# B&R Automation Studio project EFI (part 26)

#### CleaningTests.c - Groups test cases for addition
```c
/********************************************************************
 * COPYRIGHT -- Bernecker + Rainer
 ********************************************************************
 * Program: ConsentsTests
 * Author: Jorge Murria
 ********************************************************************
 * Prepare machine with basic test to allow proper behabior
 * and starting tasks
 ********************************************************************/

#include <bur/plctypes.h>

#ifdef _DEFAULT_INCLUDES
#include <AsDefault.h>
#endif

#include "UnitTest.h"

#include <stdio.h>
#include <unistd.h>
#include <time.h>         /* clock_t, clock, CLOCKS_PER_SEC */

_LOCAL TIME TimeLast;
_LOCAL TIME endtime;
_LOCAL UDINT diff_t;
_LOCAL STRING stringAux[120];

#define FALSE 0
#define TRUE 1

_LOCAL UDINT previousTileCounter;

void nextState(){
	exTimesPreFast = gMachine.St.exec.fast;
	exTimesPreSlow = gMachine.St.exec.slow;
	iTestState++;
	TimeLast = clock_ms();
	diff_t = diff_t;
	stringAux[120] = stringAux[120];
}

_TEST test_ReturningToPrint(void)
{
	strcpy(txTest, "test_ReturningToPrint");
	switch (iTestState)
	{
		case 0:
			gSimMachine.Commands.xToZero = TRUE;
			gFeeder.ParSw.xEnabled=FALSE;
			gPrimer.ParSw.xEnabled=FALSE;
			gDryerAnc.ParSw.xEnabled=FALSE;
			gStacker.ParSw.xEnabled=FALSE;
			gMachine.parSw.Media.rLength = 1600;
			gSimThickCtrl.Commands.xEmptyMediaTracking = TRUE;
			nextState();
			break;

		case 1:
			strcpy(txStateDesc, "Waiting the machine to be in Zero");
			TEST_BUSY_CONDITION( !gMachine.St.Mode.xZero );
			nextState();
			break;

		case 2:
			gSimMachine.Commands.xToAuto = TRUE;
			nextState();
			break;

		case 3:
			strcpy(txStateDesc, "Waiting the machine to be in Auto");
			TEST_BUSY_CONDITION( !gMachine.St.Mode.xAuto );
			TEST_BUSY_CONDITION( gMachine.St.exec.fast < exTimesPreFast + 8 ); //We'll wait xx scan cycles
			TEST_BUSY_CONDITION( !gMachine.St.Position.xInCap );
			gSimMachine.Commands.xToProduction = TRUE;
			nextState();
			break;

		case 4:
			strcpy(txStateDesc, "Going to Production");
			TEST_BUSY_CONDITION( !gMachine.St.AutoMode.xProduction);
			gMachine.commandsSw.xStart_GI = FALSE;
			nextState();
			break;

		case 5:
			strcpy(txStateDesc, "Waiting to be GoingToPrint");
			TEST_BUSY_CONDITION( !gMachine.St.Position.xGoingToPrint );
			TEST_BUSY_CONDITION( gBlock[1].Status.rMotorPosition > gBlock[1].parameters.Motor.rDripBarsPosition - 10);
			nextState();
			break;

		case 6:
			strcpy(txStateDesc, "Order to Clean");
			if(!gMachine.Pt.xControlledByLine ){
				gBlock[1].commands.xForceCleanNoDelay = TRUE;
			}
			else{
				gLine.Commands.Clean = TRUE;
			}
			TEST_BUSY_CONDITION( !gBlock[1].Status.Position.xCleaning);
			nextState();
			break;

		case 7:
			strcpy(txStateDesc, "Waiting to remove the signal");
			TEST_BUSY_CONDITION( gMachine.St.exec.fast < exTimesPreFast + 3 ); //We'll wait xx scan cycles
			gBlock[1].commands.xForceCleanNoDelay = FALSE;
			nextState();
			break;

		case 8:
			strcpy(txStateDesc, "Waiting to start cleaning");
			TEST_BUSY_CONDITION(gBlock[1].Status.Position.xCleaning); //We'll wait xx scan cycles
			nextState();
			break;

		case 9:
			strcpy(txStateDesc, "Waiting to finish cleaning");
			TEST_BUSY_CONDITION( gBlock[1].Status.rMotorPosition > gBlock[1].parameters.Motor.rDripBarsPosition - 10);
			nextState();
			break;

		case 10:
			endtime = clock_ms();
			TEST_BUSY_CONDITION( endtime < TimeLast + 2000 ); //We'll wait xx ms
			//TEST_ASSERT(gBlock[1].Status.Position.xGoingToPrint || gBlock[1].Status.Position.xInPrint); //If variable is TRUE, the test is correct
			TEST_ASSERT(!gBlock[1].Status.Position.xCleaning);
			nextState();
			break;

		case 11:
			strcpy(txStateDesc, "Check activation of waste ink pump");
			if(gBlock[1].parameters.xWastedInkTankProcess){
				TEST_ASSERT(gBlock[1].Out.xWastedInkTankPump);
			}

			iTestState = 0;
			TEST_DONE;

			break;

		default:
			break;
	}
}

_TEST test_ReturningToCap(void)
{
	strcpy(txTest, "test_ReturningToCap");
	switch (iTestState)
	{
		case 0:
			gSimMachine.Commands.xToZero = TRUE;
			gSimThickCtrl.Commands.xEmptyMediaTracking = TRUE;
			nextState();
			break;

		case 1:
			strcpy(txStateDesc, "Waiting the machine to be in Zero");
			TEST_BUSY_CONDITION( !gMachine.St.Mode.xZero );
			nextState();
			break;

		case 2:
			endtime = clock_ms();
			TEST_BUSY_CONDITION( endtime < TimeLast + 100 ); //We'll wait xx ms
			gSimMachine.Commands.xToAuto = TRUE;
			nextState();
			break;

		case 3:
			strcpy(txStateDesc, "Waiting the machine to be in Auto");
			TEST_BUSY_CONDITION( !gMachine.St.Mode.xAuto );
			nextState();
			break;

		case 4:
			strcpy(txStateDesc, "Waiting to be in Cap or GoingToCap");
			TEST_BUSY_CONDITION( gMachine.St.exec.fast < exTimesPreFast + 3 ); //We'll wait xx scan cycles
			TEST_BUSY_CONDITION( !gBlock[1].Status.Position.xGoingToCap  && !gBlock[1].Status.Position.xInCap);
			nextState();
			break;

		case 5:
			TEST_BUSY_CONDITION(!gBlock[1].Status.Position.xInCap);
			nextState();
			break;

		case 6:
			strcpy(txStateDesc, "Order to Clean");
			if(!gMachine.Pt.xControlledByLine ){
				gBlock[1].commands.xForceCleanNoDelay = TRUE;
			}
			else{
				gLine.Commands.Clean = TRUE;
			}
			TEST_BUSY_CONDITION( !gBlock[1].Status.Position.xCleaning); //We'll wait xx scan cycles
			nextState();
			break;

		case 7:
			strcpy(txStateDesc, "Waiting to remove the signal");
			TEST_BUSY_CONDITION( gMachine.St.exec.fast < exTimesPreFast + 3 ); //We'll wait xx scan cycles
			gBlock[1].commands.xForceCleanNoDelay = FALSE;
			nextState();
			break;

		case 8:
			strcpy(txStateDesc, "Waiting to start cleaning");
			TEST_BUSY_CONDITION( !gBlock[1].Status.Position.xCleaning); //We'll wait xx scan cycles
			nextState();
			break;

		case 9:
			strcpy(txStateDesc, "Waiting to finish cleaning");
			TEST_BUSY_CONDITION( gBlock[1].Status.Position.xCleaning); //We'll wait xx scan cycles
			nextState();
			break;

		case 10:
			TEST_BUSY_CONDITION( gMachine.St.exec.fast < exTimesPreFast + 3 ); //We'll wait xx scan cycles
			TEST_ASSERT(gBlock[1].Status.Position.xGoingToCap || gBlock[1].Status.Position.xInCap); //If variable is TRUE, the test is correct

			iTestState = 0;
			TEST_DONE;

			break;

		default:
			break;
	}
}

_TEST test_CheckAnyCleaningModeIsEnabled(void)
{
	strcpy(txTest, "test_CheckAnyCleaningModeIsEnabled");
	switch (iTestState)
	{
		case 0:
			gSimMachine.Commands.xToZero = TRUE;
			gMachine.parSw.Clean.xCleanSystemByPieces = FALSE;
			gMachine.parSw.Clean.xCleanSystemByTime = FALSE;
			gSimThickCtrl.Commands.xEmptyMediaTracking = TRUE;
			nextState();
			break;

		case 1:
			strcpy(txStateDesc, "Waiting to finish cleaning");
			TEST_BUSY_CONDITION( gMachine.St.exec.fast < exTimesPreFast + 8 ); //We'll wait xx scan cycles
			TEST_ASSERT(gMachine.Al.Warning.xNoCleaningModeEnabled); //If variable is TRUE, the test is correct

			iTestState = 0;
			TEST_DONE;

			break;

		default:
			break;
	}
}

_TEST test_CleaningByTilesTwice(void)
{
	//If the Test makes non sense, not execute it.
	if (gMachine.Pt.PDSignalTpe==PDCFG_SENSOR){

		iTestState = 0;
		TEST_DONE;
	}
	strcpy(txTest, "test_CleaningByTilesTwice");
	switch (iTestState)
	{
		case 0:
			gSimMachine.Commands.xToZero = TRUE;
			gMachine.parSw.Clean.xCleanSystemByPieces = TRUE;
			gSimMachine.Signals.xPDCarriageSignalL1 = FALSE; //To be sure to receive later the required edge
			gMachine.parSw.Clean.iPiecesNumberToCleanL1 = 10;
			gMachine.parSw.Clean.tiTimeDelayToCleanL1 = 1000;
			gMachine.parSw.Clean.tiTimeDelayGapToClean = 1000;
			gSimThickCtrl.Commands.xEmptyMediaTracking = TRUE;
			nextState();
			break;

		case 1:
			strcpy(txStateDesc, "Waiting the machine to be in Zero");
			TEST_BUSY_CONDITION( !gMachine.St.Mode.xZero );
			nextState();
			break;

		case 2:
			endtime = clock_ms();
			TEST_BUSY_CONDITION( endtime < TimeLast + 100 ); //We'll wait xx ms
			gSimMachine.Commands.xToAuto = TRUE;
			nextState();
			break;

		case 3:
			strcpy(txStateDesc, "Waiting the machine to be in Auto");
			TEST_BUSY_CONDITION( !gMachine.St.Mode.xAuto );
			nextState();
			break;

		case 4:
			strcpy(txStateDesc, "Waiting to be in Cap or GoingToCap");
			TEST_BUSY_CONDITION( gMachine.St.exec.fast < exTimesPreFast + 3 ); //We'll wait xx scan cycles
			TEST_BUSY_CONDITION( !gBlock[1].Status.Position.xGoingToCap  && !gBlock[1].Status.Position.xInCap);
			gMachine.commandsSw.xToNormal_GI = TRUE;
			nextState();
			break;

		case 5:
			strcpy(txStateDesc, "Waiting to be in Production");
			TEST_BUSY_CONDITION( !gMachine.St.AutoMode.xProduction );
			TEST_BUSY_CONDITION( gMachine.St.exec.fast < exTimesPreFast + 20 ); //We'll wait xx scan cycles
			gSimMachine.Commands.xToProduction = TRUE;
			gMachine.commandsSw.xToNormal_GI = FALSE;
			nextState();
			break;

		case 6:
			TEST_BUSY_CONDITION( gMachine.St.exec.fast < exTimesPreFast + 20 ); //We'll wait xx scan cycles
			gMachine.commandsSw.xStart_GI = FALSE;
			TEST_BUSY_CONDITION( !gBelt.states.xRuningBelt );
			previousTileCounter = gMachine.Lg.udiPiecesCounterL1;
			gDing.In.xDingLow = TRUE;
			gDing.In.rHighDingMm = 5.0;
			nextState();
			break;

		case 7:
			strcpy(txStateDesc, "Raising product detects when the belt running");
			endtime = clock_ms();
			TEST_BUSY_CONDITION( endtime < TimeLast + 200 ); //We'll wait xx ms
			if(gMachine.Pt.PDSignalTpe==PDCFG_SENSOR){
				gSimMachine.Commands.Media.xContinuousMediaPresent = TRUE;
			}
			else{
				if (previousTileCounter == gMachine.Lg.udiPiecesCounterL1) {
					gSimMachine.Signals.xPDCarriageSignalL1 = TRUE;
					gSimMachine.Signals.xProductDetectL1 = TRUE;
				}
				else {
					TimeLast = clock_ms();
					previousTileCounter = gMachine.Lg.udiPiecesCounterL1;
					gSimMachine.Signals.xPDCarriageSignalL1 = FALSE;
					gSimMachine.Signals.xProductDetectL1 = FALSE;
				}
			}
			TEST_BUSY_CONDITION( !gMachine.AutoCmd.xCleanningByPiecesL1);
			gSimMachine.Commands.Media.xContinuousMediaPresent = FALSE;
			nextState();
			break;
		case 8:
			strcpy(txStateDesc, "Waiting to start cleaning");
			gDing.In.xDingLow = FALSE;
			gDing.In.rHighDingMm = 0.0;
			TEST_BUSY_CONDITION( !gBlock[1].Status.Position.xCleaning);
			nextState();
			break;

		case 9:
			strcpy(txStateDesc, "Waiting to finish cleaning");
			TEST_BUSY_CONDITION( !gBlock[1].Status.Position.xInPrint); //We'll wait xx scan cycles
			gDing.In.xDingLow = TRUE;
			gDing.In.rHighDingMm = 5.0;
			nextState();
			break;

		case 10:
			strcpy(txStateDesc, "Raising product detects 2nd round");
			TEST_BUSY_CONDITION( !gBelt.states.xRuningBelt ); //We'll wait xx scan cycles
			endtime = clock_ms();
			TEST_BUSY_CONDITION( endtime < TimeLast + 200 ); //We'll wait xx ms
			if (previousTileCounter == gMachine.Lg.udiPiecesCounterL1) {
				gSimMachine.Signals.xPDCarriageSignalL1 = TRUE;
				gSimMachine.Signals.xProductDetectL1 = TRUE;
			}
			else {
				TimeLast = clock_ms();
				previousTileCounter = gMachine.Lg.udiPiecesCounterL1;
				gSimMachine.Signals.xPDCarriageSignalL1 = FALSE;
				gSimMachine.Signals.xProductDetectL1 = FALSE;
			}
			TEST_BUSY_CONDITION( !gMachine.AutoCmd.xCleanningByPiecesL1); //We'll wait xx scan cycles
			gSimMachine.Signals.xPDCarriageSignalL1 = FALSE;
			gSimMachine.Signals.xProductDetectL1 = FALSE;
			nextState();
			break;
		case 11:
			strcpy(txStateDesc, "Waiting to start cleaning");
			gDing.In.xDingLow = FALSE;
			gDing.In.rHighDingMm = 0.0;
			TEST_BUSY_CONDITION( !gBlock[1].Status.Position.xCleaning);
			nextState();
			break;

		case 12:
			strcpy(txStateDesc, "Waiting to finish cleaning");
			TEST_BUSY_CONDITION( gBlock[1].Status.Position.xCleaning); //We'll wait xx scan cycles
			nextState();
			break;

		case 13:
			TEST_BUSY_CONDITION( gMachine.St.exec.fast < exTimesPreFast + 5 ); //We'll wait xx scan cycles
			TEST_ASSERT(gBlock[1].Status.Position.xGoingToPrint || gBlock[1].Status.Position.xInPrint); //Prior to cleaning, it was in production, in printin
			gMachine.parSw.Clean.xCleanSystemByPieces = FALSE;
			iTestState = 0;
			TEST_DONE;

			break;

		default:
			break;
	}
}

/* --- Test for DELOREAN-2123 Cleaning belt process stopping behaviour --- */
_TEST test_CleanBeltStop(void)
{
	//If the Test makes non sense, not execute it.
	if (!gMachine.Pt.Clean.xCleanBeltForUv || !gMachine.Pt.xControlledByLine){
		//This 2 lines just for the last TestCase
		strcpy(txTest, "test_CleanBeltForUv Finished!! Congrats!");
		strcpy(txStateDesc, "--");

		iTestState = 0;
		TEST_DONE;
	}

	strcpy(txTest, "test_CleanBeltStop");
	switch (iTestState)
	{
		case 0:
			gMachine.parSw.CleanBelt.iBeltTurns = 1;
			gSimMachine.Commands.xToZero = TRUE;
			gSimThickCtrl.Commands.xEmptyMediaTracking = TRUE;
			nextState();
			break;

		case 1:
			strcpy(txStateDesc, "Waiting the machine to be in Zero");
			TEST_BUSY_CONDITION( !gMachine.St.Mode.xZero );
			nextState();
			break;

		case 2:
			TEST_BUSY_CONDITION( gMachine.St.exec.fast < exTimesPreFast + 3 ); //We'll wait xx ms
			gSimMachine.Commands.xToAuto = TRUE;
			nextState();
			break;

		case 3:
			strcpy(txStateDesc, "Waiting the machine to be in Auto");
			TEST_BUSY_CONDITION( !gMachine.St.Mode.xAuto );
			TEST_BUSY_CONDITION( gMachine.St.exec.fast < exTimesPreFast + 8 ); //We'll wait xx scan cycles
			gMachine.In.Buttons.xReset = TRUE;
			nextState();
			break;

		case 4:
			strcpy(txStateDesc, "Waiting to be in idle to send clean bealt order");
			TEST_BUSY_CONDITION (gLine.Status != LINE_IDLE);
			gMachine.commandsSw.xCleanBelt = TRUE;
			nextState();
			break;

		case 5:
			strcpy(txStateDesc, "Check belt clean process is being executed");
			TEST_BUSY_CONDITION(gMachine.St.CleaningBelt.enState != CLN_BELT_CLEAN_CLOKWISE);
			gMachine.In.Buttons.xStop = TRUE;
			nextState();
			break;

		case 6:
			strcpy(txStateDesc, "Check belt cleaning stops");
			TEST_BUSY_CONDITION( gMachine.St.exec.fast < exTimesPreFast + 5 ); //We'll wait xx scan cycles
			gMachine.In.Buttons.xStop = FALSE;
			endtime = clock_ms();
			TEST_BUSY_CONDITION( gMachine.St.CleaningBelt.enState != CLN_BELT_ERROR);// && endtime < TimeLast + 1000);
			TEST_ASSERT( gMachine.St.CleaningBelt.enState == CLN_BELT_ERROR );
			nextState();
			break;

		case 7:
			strcpy(txStateDesc, "Check belt cleaning grafcet status goes back to ready");
			endtime = clock_ms();
			TEST_BUSY_CONDITION( gMachine.St.CleaningBelt.enState != CLN_BELT_READY_TO_CLEAN);// && endtime < TimeLast + 2000);
			TEST_ASSERT( gMachine.St.CleaningBelt.enState == CLN_BELT_READY_TO_CLEAN );

			//This 2 lines just for the last TestCase
			strcpy(txTest, "test_CleaningTests Finished!! Congrats!");
			strcpy(txStateDesc, "--");

			iTestState = 0;
			TEST_DONE;

			break;

		default:
			break;
	}
}
/* --- End test for DELOREAN-2123 --- */

_TEST test_StopBelWhenMediaDetectInClean(void)
{
	strcpy(txTest, "test_StopBelWhenMediaDetectInClean");
	switch (iTestState)
	{
		case 0:
			gSimMachine.Commands.xToZero = TRUE;
			gMachine.parSw.Clean.xCleanSystemByPieces = TRUE;
			gSimMachine.Signals.xPDCarriageSignalL1 = FALSE; //To be sure to receive later the required edge
			gMachine.parSw.Clean.iPiecesNumberToCleanL1 = 10;
			gMachine.parSw.Clean.tiTimeDelayToCleanL1 = 1000;
			gMachine.parSw.Clean.tiTimeDelayGapToClean = 1000;
			gSimThickCtrl.Commands.xEmptyMediaTracking = TRUE;
			nextState();
			break;

		case 1:
			strcpy(txStateDesc, "Waiting the machine to be in Zero");
			TEST_BUSY_CONDITION( !gMachine.St.Mode.xZero );
			nextState();
			break;

		case 2:
			endtime = clock_ms();
			TEST_BUSY_CONDITION( endtime < TimeLast + 100 ); //We'll wait xx ms
			gSimMachine.Commands.xToAuto = TRUE;
			nextState();
			break;

		case 3:
			strcpy(txStateDesc, "Waiting the machine to be in Auto");
			TEST_BUSY_CONDITION( !gMachine.St.Mode.xAuto );
			nextState();
			break;

		case 4:
			strcpy(txStateDesc, "Waiting to be in Cap or GoingToCap");
			TEST_BUSY_CONDITION( gMachine.St.exec.fast < exTimesPreFast + 3 ); //We'll wait xx scan cycles
			TEST_BUSY_CONDITION( !gBlock[1].Status.Position.xGoingToCap  && !gBlock[1].Status.Position.xInCap);
			gMachine.commandsSw.xToNormal_GI = TRUE;
			nextState();
			break;

		case 5:
			strcpy(txStateDesc, "Waiting to be in Production");
			TEST_BUSY_CONDITION( !gMachine.St.AutoMode.xProduction );
			TEST_BUSY_CONDITION( gMachine.St.exec.fast < exTimesPreFast + 20 ); //We'll wait xx scan cycles
			gSimMachine.Commands.xToProduction = TRUE;
			gMachine.commandsSw.xToNormal_GI = FALSE;
			nextState();
			break;

		case 6:
			TEST_BUSY_CONDITION( gMachine.St.exec.fast < exTimesPreFast + 20 ); //We'll wait xx scan cycles
			gMachine.commandsSw.xStart_GI = FALSE;
			TEST_BUSY_CONDITION( !gBelt.states.xRuningBelt );
			previousTileCounter = gMachine.Lg.udiPiecesCounterL1;
			gDing.In.xDingLow = TRUE;
			gDing.In.rHighDingMm = 5.0;
			nextState();
			break;

		case 7:
			strcpy(txStateDesc, "Raising product detects when the belt running");
			endtime = clock_ms();
			TEST_BUSY_CONDITION( endtime < TimeLast + 200 ); //We'll wait xx ms
			if(gMachine.Pt.PDSignalTpe==PDCFG_SENSOR){
				gSimMachine.Commands.Media.xContinuousMediaPresent = TRUE;
			}
			else{
				if (previousTileCounter == gMachine.Lg.udiPiecesCounterL1) {
					gSimMachine.Signals.xPDCarriageSignalL1 = TRUE;
					gSimMachine.Signals.xProductDetectL1 = TRUE;
				}
				else {
					TimeLast = clock_ms();
					previousTileCounter = gMachine.Lg.udiPiecesCounterL1;
					gSimMachine.Signals.xPDCarriageSignalL1 = FALSE;
					gSimMachine.Signals.xProductDetectL1 = FALSE;
				}
			}
			TEST_BUSY_CONDITION( !gMachine.AutoCmd.xCleanningByPiecesL1);
			gSimMachine.Commands.Media.xContinuousMediaPresent = FALSE;
			nextState();
			break;
		case 8:
			strcpy(txStateDesc, "Waiting to start cleaning");
			gDing.In.xDingLow = FALSE;
			gDing.In.rHighDingMm = 0.0;
			gPhotoCells.Inputs.Signals.xPhotoCells[1] = FALSE;
			TEST_BUSY_CONDITION( !gBlock[1].Status.Position.xCleaning);
			nextState();
			break;

		case 9:
			strcpy(txStateDesc, "Detect Media In");
			if (gDing.State.xDingInstalled){
				gDing.In.xDingLow = TRUE;
				gDing.In.rHighDingMm = 5.0;
			}
			else{
				gPhotoCells.Inputs.Signals.xPhotoCells[1] = TRUE;
			}
			nextState();
			break;

		case 10:
			TEST_BUSY_CONDITION( gMachine.St.exec.fast < exTimesPreFast + 10 ); //We'll wait xx scan cycles
			TEST_ASSERT(!gBelt.states.xRuningBelt); //Prior to cleaning, it was in production, in printing
			nextState();
			break;

		case 11:
			strcpy(txStateDesc, "Waiting to finish cleaning");
			TEST_BUSY_CONDITION( gBlock[1].Status.Position.xCleaning); //We'll wait xx scan cycles
			gMachine.parSw.Clean.xCleanSystemByPieces = FALSE;
			gDing.In.xDingLow = FALSE;
			gPhotoCells.Inputs.Signals.xPhotoCells[1] = FALSE;
			//This 2 lines just for the last TestCase
			strcpy(txTest, "test_CleaningTests Finished!! Congrats!");
			strcpy(txStateDesc, "--");
			iTestState = 0;
			TEST_DONE;

			break;

		default:
			break;

//		case 12:
//			TEST_BUSY_CONDITION( gMachine.St.exec.fast < exTimesPreFast + 5 ); //We'll wait xx scan cycles
//			TEST_ASSERT(gBlock[1].Status.Position.xGoingToPrint || gBlock[1].Status.Position.xInPrint); //Prior to cleaning, it was in production, in printing
//			gMachine.parSw.Clean.xCleanSystemByPieces = FALSE;
//			//This 2 lines just for the last TestCase
//			strcpy(txTest, "test_CleaningTests Finished!! Congrats!");
//			strcpy(txStateDesc, "--");
//			iTestState = 0;
//			TEST_DONE;

//			break;

//		default:
//			break;

	}
}

_TEST test_StopVenturiWhenCloseToEnd(void)
{
	strcpy(txTest, "test_StopVenturiWhenCloseToEnd");
	switch (iTestState)
	{
		case 0:
			strcpy(txStateDesc, "Preparing test conditions...");
			gSimMachine.Commands.xToZero = TRUE;
			gSimThickCtrl.Commands.xEmptyMediaTracking = TRUE;
			nextState();
			break;

		case 1:
			TEST_BUSY_CONDITION (!gMachine.St.Mode.xZero);
			gSimMachine.Commands.xToAuto = TRUE;
			nextState();
			break;

		case 2:
			TEST_BUSY_CONDITION (!gMachine.St.Mode.xAuto);
			TEST_BUSY_CONDITION( !gBlock[1].Status.Position.xInCap);
			nextState();
			break;

		case 3:
			strcpy(txStateDesc, "Giving clean order...");
			TEST_BUSY_CONDITION ( gMachine.St.exec.fast < exTimesPreFast + 20 );
			gMachine.commands.xClean = TRUE;
			nextState();
			break;

		case 4:
			strcpy(txStateDesc, "Waiting for clean procss...");
			TEST_BUSY_CONDITION (!gBlock[1].Status.Position.xCleaning);
			TEST_BUSY_CONDITION (!gBlock[1].Status.Icla.xIsMoving);
			nextState();
			break;

		case 5:
			strcpy(txStateDesc, "Venturi should turn on");
			TEST_BUSY_CONDITION ( gBlock[1].Status.Icla.rCurrentPosition <= gBlock[1].parameters.Icla.rLastHeadPosition);
			nextState();
			break;

		case 6:
			TEST_BUSY_CONDITION ( gBlock[1].Status.Icla.rCurrentPosition >= (gBlock[1].parameters.Icla.rLastHeadPosition));
			nextState();
			break;

		case 7:
			TEST_BUSY_CONDITION(gMachine.St.exec.slow < exTimesPreSlow +3);
			TEST_ASSERT(gBlock[1].Out.xVenturi);
			nextState();
			break;

		case 8:
			strcpy(txStateDesc, "Venturi should turn off");
			TEST_BUSY_CONDITION ( gBlock[1].Status.Icla.rCurrentPosition >= gBlock[1].parameters.Icla.rFirstHeadPosition);
			nextState();
			break;

		case 9:
			TEST_BUSY_CONDITION ( gMachine.St.exec.slow < exTimesPreSlow + 3);
			TEST_ASSERT (!gBlock[1].Out.xVenturi);
			nextState();
			break;

		case 10:
			strcpy(txTest, "Waiting stop cleaning...");
			TEST_BUSY_CONDITION(gMachine.St.Cleaning.enCleaningState != CLN_NOT_CLEANING);
			TEST_BUSY_CONDITION(!gBlock[1].Status.Position.xInCap);
			nextState();

		case 11:
			strcpy(txTest, "test_CleaningTests finished");
			strcpy(txStateDesc, "--");
			iTestState = 0;
			TEST_DONE;
			break;

		default:
			break;

	}
}

_TEST test_CleanBeltForUv(void)
{
	//If the Test makes non sense, not execute it.
	if (!gMachine.Pt.Clean.xCleanBeltForUv){
		//This 2 lines just for the last TestCase
		strcpy(txTest, "test_CleanBeltForUv Finished!! Congrats!");
		strcpy(txStateDesc, "--");

		iTestState = 0;
		TEST_DONE;
	}

	strcpy(txTest, "test_CleanBeltForUv");
	switch (iTestState)
	{
		case 0:
			gSimMachine.Commands.xToZero = TRUE;
			gMachine.parSw.CleanBelt.tiCleaningBeltByTime = 60000; //1 minute
			gMachine.parSw.CleanBelt.xCleanBeltByTime = TRUE;
			gMachine.parSw.CleanBelt.iBeltSpeed = gMachine.parSw.rBeltSpeedSetPoint + 5.0;
			gMachine.parSw.CleanBelt.iBeltTurns = 2;
			gMachine.In.CleanBelt.xOpenGuide = FALSE;
			gSimThickCtrl.Commands.xEmptyMediaTracking = TRUE;
			nextState();
			break;

		case 1:
			strcpy(txStateDesc, "Waiting the machine to be in Zero");
			TEST_BUSY_CONDITION( !gMachine.St.Mode.xZero );
			nextState();
			break;

		case 2:
			TEST_BUSY_CONDITION( gMachine.St.exec.fast < exTimesPreFast + 3 ); //We'll wait xx ms
			gSimMachine.Commands.xToAuto = TRUE;
			nextState();
			break;

		case 3:
			strcpy(txStateDesc, "Waiting the machine to be in Auto");
			TEST_BUSY_CONDITION( !gMachine.St.Mode.xAuto );
			nextState();
			break;

		case 4:
			strcpy(txStateDesc, "Waiting to be in Cap or GoingToCap");
			TEST_BUSY_CONDITION( gMachine.St.exec.fast < exTimesPreFast + 3 ); //We'll wait xx scan cycles
			TEST_BUSY_CONDITION( !gBlock[1].Status.Position.xGoingToCap  && !gBlock[1].Status.Position.xInCap);
			gMachine.commandsSw.xToNormal_GI = TRUE;
			nextState();
			break;

		case 5:
			strcpy(txStateDesc, "Waiting to be in Production");
			TEST_BUSY_CONDITION( !gMachine.St.AutoMode.xProduction );
			TEST_BUSY_CONDITION( gMachine.St.exec.fast < exTimesPreFast + 20 ); //We'll wait xx scan cycles
			gSimMachine.Commands.xToProduction = TRUE;
			TEST_BUSY_CONDITION( !gBelt.states.xRuningBelt );
			nextState();
			break;

		case 6:
			TEST_BUSY_CONDITION( gMachine.St.exec.fast < exTimesPreFast + 20 ); //We'll wait xx scan cycles
			endtime = clock_ms();
			TEST_BUSY_CONDITION( endtime <= TimeLast + gMachine.parSw.CleanBelt.tiCleaningBeltByTime*2 ); //We'll wait xx ms
			nextState();
			break;

		case 7:
			strcpy(txStateDesc, "Waiting to be in Production");
			TEST_BUSY_CONDITION( gMachine.St.exec.fast < exTimesPreFast + 20 ); //We'll wait xx scan cycles
			if(!gMachine.Pt.xControlledByLine ){
				gMachine.commandsSw.xStop_GI = TRUE;
			}
			else{
				gLine.Commands.Stop = TRUE;
			}
			nextState();
			break;

		case 8:
			strcpy(txStateDesc, "Waiting to be ready to clean");
			TEST_BUSY_CONDITION(gBelt.states.xRuningBelt);
			if(!gMachine.Pt.xControlledByLine ){
			TEST_BUSY_CONDITION(!gMachine.St.AutoMode.xStop);
			}
			else{
			TEST_BUSY_CONDITION(!gLine.StatusSummary.xIdle);
			}
			TEST_BUSY_CONDITION(!gMachine.St.CleaningBelt.xCleanRequired); //We'll wait xx scan cycles
			TEST_ASSERT(gMachine.St.CleaningBelt.xCleanRequired);
			nextState();
			break;

		/* Test to check disable belt clean motor neumatic movements if cleaning system is out DELOREAN-1606 */
		case 9:
			strcpy(txStateDesc, "Send clean belt order");
			gMachine.commandsSw.xCleanBelt = TRUE;
			TEST_BUSY_CONDITION(!gMachine.AutoCmd.xCleanBelt); //We'll wait xx scan cycles
			TEST_ASSERT(gMachine.AutoCmd.xCleanBelt);
			nextState();
			break;

		case 10:
			strcpy(txStateDesc, "Check belt clean process is being executed");
			TEST_BUSY_CONDITION(!gMachine.St.CleaningBelt.xCleaningProcessOnGoing); //We'll wait xx scan cycles
			gMachine.commandsSw.xCleanBelt = FALSE;
			TEST_ASSERT(gMachine.St.CleaningBelt.xCleaningProcessOnGoing);
			TEST_ASSERT(gBelt.parameters.rSetPointSpeed=gMachine.parSw.CleanBelt.iBeltSpeed);
			nextState();
			break;

		/* Test to check delay on swaping clean belt motor direction DELOREAN-1607 */
		case 11:
			strcpy(txStateDesc, "Check belt clean motor moves forward");
			TEST_BUSY_CONDITION(!gMachine.commands.CleanBelt.xCleanBeltMoveFwd);
			TEST_ASSERT(gMachine.commands.CleanBelt.xCleanBeltMoveFwd );
			TEST_ASSERT(!gMachine.commands.CleanBelt.xCleanBeltMoveBwd );
			nextState();
			break;

		case 12:
			strcpy(txStateDesc, "Check belt clean motor stops");
			TEST_BUSY_CONDITION(gMachine.commands.CleanBelt.xCleanBeltMoveFwd);
			TEST_ASSERT(!gMachine.commands.CleanBelt.xCleanBeltMoveFwd );
			TEST_ASSERT(!gMachine.commands.CleanBelt.xCleanBeltMoveBwd );
			nextState();
			break;

		case 13:
			strcpy(txStateDesc, "Check belt clean motor moves backward");
			endtime = clock_ms();
			TEST_BUSY_CONDITION( endtime < TimeLast + 4000 );
			TEST_ASSERT(gMachine.commands.CleanBelt.xCleanBeltMoveFwd );
			TEST_ASSERT(!gMachine.commands.CleanBelt.xCleanBeltMoveBwd );
			nextState();
			break;

		case 14:
			strcpy(txStateDesc, "Check belt clean motor stops");
			TEST_BUSY_CONDITION(gMachine.commands.CleanBelt.xCleanBeltMoveFwd);
			TEST_ASSERT(!gMachine.commands.CleanBelt.xCleanBeltMoveFwd );
			TEST_ASSERT(!gMachine.commands.CleanBelt.xCleanBeltMoveBwd );
			nextState();
			break;

		case 15:
			strcpy(txStateDesc, "Check belt clean motor moves backward");
			endtime = clock_ms();
			TEST_BUSY_CONDITION( endtime < TimeLast + gMachine.St.CleaningBelt.TimeDelaySwapDirBeltCleanMotor + 250 );
			TEST_ASSERT(!gMachine.commands.CleanBelt.xCleanBeltMoveFwd );
			TEST_ASSERT(gMachine.commands.CleanBelt.xCleanBeltMoveBwd );
			nextState();
			break;

		case 16:
			strcpy(txStateDesc, "Check belt is stopped");
			TEST_BUSY_CONDITION(gMachine.St.CleaningBelt.xCleaningProcessOnGoing);
			TEST_ASSERT(!gMachine.commands.xRunBelt); //If variable is TRUE, the test is correct
			gMachine.parSw.CleanBelt.xCleanBeltByTime = FALSE;

			iTestState = 0;
			TEST_DONE;

			break;

		default:
			break;
	}
}

//DELOREAN-1606
_TEST test_CleanBeltForUvIsNotExecutedWhenGuideIsOpened(void)
{
	//If the Test makes non sense, not execute it.
	if (!gMachine.Pt.Clean.xCleanBeltForUv){
		//This 2 lines just for the last TestCase
		strcpy(txTest, "test_CleanBeltForUvIsNotExecutedWhenGuideIsOpened Finished!! Congrats!");
		strcpy(txStateDesc, "--");

		iTestState = 0;
		TEST_DONE;
	}

	strcpy(txTest, "test_CleanBeltForUvIsNotExecutedWhenGuideIsOpened");
	switch (iTestState)
	{
		case 0:
			gSimMachine.Commands.xToZero = TRUE;
			gMachine.parSw.CleanBelt.tiCleaningBeltByTime = 60000; //1 minute
			gMachine.parSw.CleanBelt.xCleanBeltByTime = TRUE;
			gMachine.parSw.CleanBelt.iBeltSpeed = gMachine.parSw.rBeltSpeedSetPoint + 5.0;
			gMachine.parSw.CleanBelt.iBeltTurns = 2;
			gSimThickCtrl.Commands.xEmptyMediaTracking = TRUE;
			nextState();
			break;

		case 1:
			strcpy(txStateDesc, "Waiting the machine to be in Zero");
			TEST_BUSY_CONDITION( !gMachine.St.Mode.xZero );
			nextState();
			break;

		case 2:
			TEST_BUSY_CONDITION( gMachine.St.exec.fast < exTimesPreFast + 3 ); //We'll wait xx ms
			gSimMachine.Commands.xToAuto = TRUE;
			nextState();
			break;

		case 3:
			strcpy(txStateDesc, "Waiting the machine to be in Auto");
			TEST_BUSY_CONDITION( !gMachine.St.Mode.xAuto );
			nextState();
			break;

		case 4:
			strcpy(txStateDesc, "Waiting to be in Cap or GoingToCap");
			TEST_BUSY_CONDITION( gMachine.St.exec.fast < exTimesPreFast + 3 ); //We'll wait xx scan cycles
			TEST_BUSY_CONDITION( !gBlock[1].Status.Position.xGoingToCap  && !gBlock[1].Status.Position.xInCap);
			gMachine.commandsSw.xToNormal_GI = TRUE;
			nextState();
			break;

		case 5:
			strcpy(txStateDesc, "Waiting to be in Production");
			TEST_BUSY_CONDITION( !gMachine.St.AutoMode.xProduction );
			TEST_BUSY_CONDITION( gMachine.St.exec.fast < exTimesPreFast + 20 ); //We'll wait xx scan cycles
			gSimMachine.Commands.xToProduction = TRUE;
			TEST_BUSY_CONDITION( !gBelt.states.xRuningBelt );
			nextState();
			break;

		case 6:
			TEST_BUSY_CONDITION( gMachine.St.exec.fast < exTimesPreFast + 20 ); //We'll wait xx scan cycles
			endtime = clock_ms();
			TEST_BUSY_CONDITION( endtime <= TimeLast + gMachine.parSw.CleanBelt.tiCleaningBeltByTime*2 ); //We'll wait xx ms
			nextState();
			break;

		case 7:
			strcpy(txStateDesc, "Waiting to be in Production");
			TEST_BUSY_CONDITION( gMachine.St.exec.fast < exTimesPreFast + 20 ); //We'll wait xx scan cycles
			if(!gMachine.Pt.xControlledByLine ){
				gMachine.commandsSw.xStop_GI = TRUE;
			}
			else{
				gLine.Commands.Stop = TRUE;
			}
			gMachine.In.CleanBelt.xOpenGuide = TRUE;
			nextState();
			break;

		case 8:
			strcpy(txStateDesc, "Waiting to be ready to clean");
			TEST_BUSY_CONDITION(gBelt.states.xRuningBelt);
			if(!gMachine.Pt.xControlledByLine ){
				TEST_BUSY_CONDITION(!gMachine.St.AutoMode.xStop);
			}
			else{
				TEST_BUSY_CONDITION(!gLine.StatusSummary.xIdle);
			}
			//			TEST_BUSY_CONDITION(!gMachine.St.CleaningBelt.xCleanRequired);
			nextState();
			break;

		case 9:
			strcpy(txStateDesc, "Send clean belt order with blockage of clean belt motor position");
			gMachine.commandsSw.xCleanBelt = TRUE;
			TEST_BUSY_CONDITION(!gMachine.AutoCmd.xCleanBelt); //We'll wait xx scan cycles
			nextState();
			break;

		case 10:
			strcpy(txStateDesc, "Check if alarm is displayed and clean motor moved");
			TEST_BUSY_CONDITION( gMachine.St.exec.fast < exTimesPreFast + 8 );
			TEST_ASSERT(gMachine.Al.Warning.xCleanBeltSystemNotInPosition);
			TEST_ASSERT(!gMachine.commands.CleanBelt.xPistonFlojet);
			TEST_ASSERT(!gMachine.St.CleaningBelt.xCleanRequired);
			gMachine.In.CleanBelt.xOpenGuide = FALSE;
			nextState();
			break;

		case 11:
			strcpy(txStateDesc, "Check belt is stopped");
			TEST_BUSY_CONDITION(!gMachine.St.CleaningBelt.xCleaningProcessOnGoing);
			TEST_ASSERT(gMachine.commands.xRunBelt);
			gMachine.parSw.CleanBelt.xCleanBeltByTime = FALSE;

			strcpy(txTest, "CleaningTests Finished!! Congrats!");
			strcpy(txStateDesc, "--");

			iTestState = 0;
			TEST_DONE;

			break;

		default:
			break;
	}
}

/*
B+R UnitTest: This is generated code.
Do not edit! Do not move!
Description: UnitTest Testprogramm infrastructure (TestSet).
LastUpdated: 2023-05-22 13:38:39Z
By B+R UnitTest Helper Version: 2.0.1.59
*/
UNITTEST_FIXTURES(fixtures)
{
	new_TestFixture("test_ReturningToPrint", test_ReturningToPrint),
	new_TestFixture("test_ReturningToCap", test_ReturningToCap),
	new_TestFixture("test_CheckAnyCleaningModeIsEnabled", test_CheckAnyCleaningModeIsEnabled),
	new_TestFixture("test_CleaningByTilesTwice", test_CleaningByTilesTwice),
	new_TestFixture("test_CleanBeltStop", test_CleanBeltStop),
	new_TestFixture("test_StopBelWhenMediaDetectInClean", test_StopBelWhenMediaDetectInClean),
	new_TestFixture("test_StopVenturiWhenCloseToEnd", test_StopVenturiWhenCloseToEnd),
	new_TestFixture("test_CleanBeltForUv", test_CleanBeltForUv),
	new_TestFixture("test_CleanBeltForUvIsNotExecutedWhenGuideIsOpened", test_CleanBeltForUvIsNotExecutedWhenGuideIsOpened),
};

UNITTEST_CALLER_COMPLETE_EXPLICIT(CleaningTests, "CleaningTests", 0, 0, fixtures, 0, 0, 0);
```

- Update_TestPrograms_in_current_location.bat - Updates test programs within the current package (not shown)

### Program Logical/UnitTest/Tests/TrVacuumTests (ANSIC)

#### TrVacuumTests.c - Groups test cases for addition
```c
/********************************************************************
 * COPYRIGHT -- Bernecker + Rainer
 ********************************************************************
 * Program: VacuumTests
 * Author: Jorge Murria
 ********************************************************************
 * Prepare machine with basic test to allow proper behabior
 * and starting tasks
 ********************************************************************/

#include <bur/plctypes.h>

#ifdef _DEFAULT_INCLUDES
#include <AsDefault.h>
#endif

#include "UnitTest.h"

#include <stdio.h>
#include <unistd.h>
#include <time.h>         /* clock_t, clock, CLOCKS_PER_SEC */

_LOCAL TIME TimeLast;
_LOCAL TIME endtime;
_LOCAL UDINT diff_t;
_LOCAL STRING stringAux[120];

#define FALSE 0
#define TRUE 1

void nextState(){
	exTimesPreFast = gMachine.St.exec.fast;
	exTimesPreSlow = gMachine.St.exec.slow;
	iTestState++;
	TimeLast = clock_ms();
	diff_t = diff_t;
	stringAux[120] = stringAux[120];
}

_TEST test_StopBlowersOutProductionByPass(void)
{
	if (!gMachine.Pt.xAllowLaboratory){
		TEST_DONE;
	}
	strcpy(txTest, "test_StopBlowersOutProduction-ByPass");
	switch (iTestState)
	{
		case 0:
			if (!gTransVacuum[1].Status.xInstalled)
			{
				TEST_DONE;
				break;
			}
			else
			{
				nextState();
				break;
			}
		case 1:
			gSimMachine.Commands.xToZero = TRUE;
			nextState();
			break;

		case 2:
			strcpy(txStateDesc, "Waiting the machine to be in Zero");
			TEST_BUSY_CONDITION( !gMachine.St.Mode.xZero );
			gTransVacuum[1].parSw.xActiveOutOfProduction = FALSE;
			gSimMachine.Commands.xToAuto = TRUE;
			gMachine.parSw.rBeltSpeedSetPoint = 70.0;
			nextState();
			break;

		case 3:
			strcpy(txStateDesc, "Waiting the machine to be in Auto");
			TEST_BUSY_CONDITION( !gMachine.St.Mode.xAuto );
			nextState();
			break;

		case 4:
			strcpy(txStateDesc, "Waiting the Belt to Start. In ByPass");
			TEST_BUSY_CONDITION( gMachine.St.exec.fast < exTimesPreFast + 3 ); //We'll wait xx scan cycles
			gMachine.commandsSw.xToByPass_GI = TRUE;
			TEST_BUSY_CONDITION(!gMachine.St.AutoMode.xBypass); //We'll wait xx scan cycles
			TEST_BUSY_CONDITION(!gBelt.states.xRuningBelt); //We'll wait xx scan cycles
			nextState();
			break;
		case 5:
			strcpy(txStateDesc, "CheckVacuumStopState");
			TEST_BUSY_CONDITION( gMachine.St.exec.fast < exTimesPreFast + 5 ); //We'll wait xx scan cycles
			TEST_ASSERT(!gTransVacuum[1].Status.Blower.rDutyCycle>0.0);

			iTestState = 0;

			TEST_DONE;
			break;

		default:
			break;
	}
}

_TEST test_StartBlowersOutProductionByPass(void)
{
	strcpy(txTest, "test_StartBlowersOutProduction-ByPass");
	switch (iTestState)
	{
		case 0:
			if (!gTransVacuum[1].Status.xInstalled)
			{
				TEST_DONE;
				break;
			}
			else
			{
				nextState();
				break;
			}

		case 1:
			gSimMachine.Commands.xToZero = TRUE;
			nextState();
			break;

		case 2:
			strcpy(txStateDesc, "Waiting the machine to be in Zero");
			TEST_BUSY_CONDITION( !gMachine.St.Mode.xZero );
			gTransVacuum[1].parSw.xActiveOutOfProduction = TRUE;
			gSimMachine.Commands.xToAuto = TRUE;
			gMachine.parSw.rBeltSpeedSetPoint = 70.0;
			nextState();
			break;

		case 3:
			strcpy(txStateDesc, "Waiting the machine to be in Auto");
			TEST_BUSY_CONDITION( !gMachine.St.Mode.xAuto );
			nextState();
			break;

		case 4:
			strcpy(txStateDesc, "Waiting the Belt to Start. In ByPass");
			TEST_BUSY_CONDITION( gMachine.St.exec.fast < exTimesPreFast + 3 ); //We'll wait xx scan cycles
			gMachine.commandsSw.xToByPass_GI = TRUE;
			TEST_BUSY_CONDITION(!gMachine.St.AutoMode.xBypass); //We'll wait xx scan cycles
			TEST_BUSY_CONDITION(!gBelt.states.xRuningBelt); //We'll wait xx scan cycles
			nextState();
			break;
		case 5:
			strcpy(txStateDesc, "CheckVacuumStopState");
			TEST_BUSY_CONDITION( gMachine.St.exec.fast < exTimesPreFast + 5 ); //We'll wait xx scan cycles
			TEST_ASSERT(gTransVacuum[1].Status.Blower.rDutyCycle>0.0);

			iTestState = 0;

			TEST_DONE;
			break;

		default:
			break;
	}
}

_TEST test_StopBlowersOutProductionLab(void)
{
	//Machines controlled by line do not have laboratory mode
	if (!gTransVacuum[1].Status.xInstalled || !gMachine.Pt.xAllowLaboratory)
	{
		TEST_DONE;
	}

	strcpy(txTest, "test_StopBlowersOutProductionLab");
	switch (iTestState)
	{
		case 0:
			//Here was previously code. Leaved like this to avoid renaming cases
			nextState();
			break;
		case 1:
			gSimMachine.Commands.xToZero = TRUE;
			nextState();
			break;

		case 2:
			strcpy(txStateDesc, "Waiting the machine to be in Zero");
			TEST_BUSY_CONDITION( !gMachine.St.Mode.xZero );
			gTransVacuum[1].parSw.xActiveOutOfProduction = FALSE;
			gSimMachine.Commands.xToAuto = TRUE;
			gMachine.parSw.rBeltSpeedSetPoint = 70.0;
			nextState();
			break;

		case 3:
			strcpy(txStateDesc, "Waiting the machine to be in Auto");
			TEST_BUSY_CONDITION( !gMachine.St.Mode.xAuto );
			nextState();
			break;

		case 4:
			strcpy(txStateDesc, "Waiting the machine in Lab");
			TEST_BUSY_CONDITION( gMachine.St.exec.fast < exTimesPreFast + 3 ); //We'll wait xx scan cycles
			gMachine.commandsSw.xToLaboratory_GI = TRUE;
			TEST_BUSY_CONDITION(!gMachine.St.AutoMode.xLaboratory); //We'll wait xx scan cycles
			nextState();
			break;

		case 5:
			strcpy(txStateDesc, "CheckVacuumStopStateStopedBelt");
			TEST_BUSY_CONDITION( gMachine.St.exec.fast < exTimesPreFast + 5 ); //We'll wait xx scan cycles
			TEST_ASSERT(!gTransVacuum[1].Status.Blower.rDutyCycle>0.0);
			gMachine.commands.xRunBelt = TRUE;
			nextState();
			break;

		case 6:
			strcpy(txStateDesc, "WaitBeltStart");
			TEST_BUSY_CONDITION( gBelt.states.xRuningBelt );
			nextState();
			break;

		case 7:
			strcpy(txStateDesc, "CheckVacuumStopStateRunningBelt");
			TEST_ASSERT(!gTransVacuum[1].Status.Blower.rDutyCycle>0.0);

			iTestState = 0;

			TEST_DONE;
			break;

		default:
			break;
	}
}

_TEST test_StartBlowersOutProductionLab(void)
{
	//Machines controlled by line do not have laboratory mode
	if (!gTransVacuum[1].Status.xInstalled || !gMachine.Pt.xAllowLaboratory)
	{
		strcpy(txTest, "test_TrVacuum Finished!! Congrats!");
		strcpy(txStateDesc, "--");
		TEST_DONE;
	}

	strcpy(txTest, "test_StartBlowersOutProductionLabLab");
	switch (iTestState)
	{
		case 0:
			//Here was previously code. Leaved like this to avoid renaming cases
			nextState();
			break;
		case 1:
			gSimMachine.Commands.xToZero = TRUE;
			nextState();
			break;

		case 2:
			strcpy(txStateDesc, "Waiting the machine to be in Zero");
			TEST_BUSY_CONDITION( !gMachine.St.Mode.xZero );
			gTransVacuum[1].parSw.xActiveOutOfProduction = TRUE;
			gSimMachine.Commands.xToAuto = TRUE;
			gMachine.parSw.rBeltSpeedSetPoint = 70.0;
			nextState();
			break;

		case 3:
			strcpy(txStateDesc, "Waiting the machine to be in Auto");
			TEST_BUSY_CONDITION( !gMachine.St.Mode.xAuto );
			nextState();
			break;

		case 4:
			strcpy(txStateDesc, "Waiting the machine in Lab");
			TEST_BUSY_CONDITION( gMachine.St.exec.fast < exTimesPreFast + 3 ); //We'll wait xx scan cycles
			gMachine.commandsSw.xToLaboratory_GI = TRUE;
			TEST_BUSY_CONDITION(!gMachine.St.AutoMode.xLaboratory); //We'll wait xx scan cycles
			nextState();
			break;

		case 5:
			strcpy(txStateDesc, "CheckVacuumStopStateStopedBelt");
			TEST_BUSY_CONDITION( gMachine.St.exec.fast < exTimesPreFast + 10 ); //We'll wait xx scan cycles
			TEST_ASSERT(!gTransVacuum[1].Status.Blower.rDutyCycle>0.0);
			gSimMachine.Commands.xToProduction = TRUE;
			nextState();
			break;

		case 6:
			strcpy(txStateDesc, "WaitBeltStart");
			TEST_BUSY_CONDITION(!gBelt.states.xRuningBelt );
			nextState();
			break;

		case 7:
			strcpy(txStateDesc, "CheckVacuumStopStateRunningBelt");
			TEST_ASSERT(gTransVacuum[1].Status.Blower.rDutyCycle>0.0);

			iTestState = 0;

			strcpy(txTest, "test_TrVacuum Finished!! Congrats!");
			strcpy(txStateDesc, "--");

			TEST_DONE;
			break;

		default:
			break;
	}
}

_TEST test_StopBlowersWhenGoingOutOfManual(void)
{
	strcpy(txTest, "test_StopBlowersWhenGoingOutOfManual");
	switch (iTestState)
	{
		case 0:
			if (!gTransVacuum[1].Status.xInstalled)
			{
				TEST_DONE;
				break;
			}
			else
			{
				nextState();
				break;
			}

		case 1:
			gSimMachine.Commands.xToManual = TRUE;
			gTransVacuum[1].parSw.rManSetPoint = 50.0;
			nextState();
			break;

		case 2:
			strcpy(txStateDesc, "Waiting the machine to be in manual");
			TEST_BUSY_CONDITION( !gMachine.St.Mode.xManual );
			gTransVacuum[1].OrdersSw.xRunManual = TRUE;
			nextState();
			break;

		case 3:
			strcpy(txStateDesc, "Waiting the blowers to be running");
			TEST_BUSY_CONDITION( !gTransVacuum[1].Status.xStartedMan );
			TEST_BUSY_CONDITION( gTransVacuum[1].Status.Blower.rDutyCycle<gTransVacuum[1].parSw.rManSetPoint );
			nextState();
			break;

		case 4:
			strcpy(txStateDesc, "Waiting the Belt to Start. In ByPass");
			gSimMachine.Commands.xToZero = TRUE;
			TEST_BUSY_CONDITION( !gMachine.St.Mode.xZero );
			nextState();
			break;

		case 5:
			strcpy(txStateDesc, "CheckVacuumStopState");
			TEST_BUSY_CONDITION( gMachine.St.exec.fast < exTimesPreFast + 5 ); //We'll wait xx scan cycles
			TEST_ASSERT(!gTransVacuum[1].Status.xStartedMan);

			iTestState = 0;

			TEST_DONE;
			break;

		default:
			break;
	}
}

_TEST test_StopBlowersWithAlarmLaboratory(void)
{
	strcpy(txTest, "test_StopBlowersWithAlarmLaboratory");
	switch (iTestState)
	{
		case 0:
			strcpy(txStateDesc, "Checking the blowers are installed");
			if ((!gTransVacuum[1].Status.xInstalled) || (!gMachine.Pt.xAllowLaboratory)){
			TEST_DONE;
			break;
			}

			else{
			strcpy(txStateDesc, "Going to ZERO");
			TEST_BUSY_CONDITION( gMachine.St.exec.fast < exTimesPreFast + 3 ); //We'll wait xx scan cycles
			gSimMachine.Commands.xToZero = TRUE;
			nextState();
			break;
			}

		case 1:
			strcpy(txStateDesc, "Waiting the machine to be in Zero");
			TEST_BUSY_CONDITION( !gMachine.St.Mode.xZero );
			gTransVacuum[1].parSw.xActiveOutOfProduction = TRUE;
			gSimMachine.Commands.xToAuto = TRUE;
			nextState();
			break;

		case 2:
			strcpy(txStateDesc, "Waiting the machine to be in Auto and CAP");
			TEST_BUSY_CONDITION(!gMachine.St.Mode.xAuto);
			TEST_BUSY_CONDITION(!gMachine.St.Position.xInCap);
			gMachine.commandsSw.xToLaboratory_GI = TRUE;
			nextState();
			break;

		case 3:
			strcpy(txStateDesc, "TEST 1: Laboratory");
			endtime = clock_ms();
			TEST_BUSY_CONDITION(endtime < TimeLast + 1000);
			nextState();
			break;

		case 4:
			strcpy(txStateDesc, "Waiting for LABORATORY mode");
			TEST_BUSY_CONDITION(!gMachine.St.AutoMode.xLaboratory);

			nextState();
			break;

		case 5:
			strcpy(txStateDesc, "Giving xStart command");
			TEST_BUSY_CONDITION( gMachine.St.exec.fast < exTimesPreFast + 3 ); //We'll wait xx scan cycles
			gMachine.commandsSw.xStart_GI = TRUE;
			nextState();
			break;

		case 6: //checking if the machine reaches the positions it has to
			strcpy(txStateDesc, "Waiting for the start process to complete");
			TEST_BUSY_CONDITION(!gMachine.St.AutoMode.xProdORLab);//averiguar cuales son las variables a comprobar
			TEST_BUSY_CONDITION(!gBelt.states.xRuningBelt);
			nextState();
			break;

		case 7:
			strcpy(txStateDesc, "BlowersStartInAOP");
			endtime=clock_ms();
			TEST_BUSY_CONDITION(endtime < TimeLast + 50);
			TEST_ASSERT(gTransVacuum[1].Status.Blower.rDutyCycle > 0);//de momento la condición no se cumple, revisar

			nextState();
			break;

		case 8:
			TEST_BUSY_CONDITION( gMachine.St.exec.fast < exTimesPreFast + 3 ); //We'll wait xx scan cycles
			gTransVacuum[1].parSw.xActiveOutOfProduction = FALSE;
			nextState();
			break;

		case 9:
			TEST_BUSY_CONDITION(gTransVacuum[1].parSw.xActiveOutOfProduction);
			nextState();
			break;

		case 10:
			endtime=clock_ms();
			TEST_BUSY_CONDITION(endtime < TimeLast + 5000);
			TEST_ASSERT(!gTransVacuum[1].Status.Blower.xMoving);
			nextState();
			break;

		case 11:
			TEST_BUSY_CONDITION( gMachine.St.exec.fast < exTimesPreFast + 3 ); //We'll wait xx scan cycles
			gTransVacuum[1].parSw.xActiveOutOfProduction = TRUE;
			gMachine.commandsSw.xStart_GI = TRUE;
			nextState();
			break;

		case 12:
			TEST_BUSY_CONDITION(!gMachine.commandsSw.xStart_GI);
			TEST_BUSY_CONDITION(!gTransVacuum[1].parSw.xActiveOutOfProduction);
			nextState();
			break;

		case 13:
			endtime=clock_ms();
			TEST_BUSY_CONDITION(endtime < TimeLast + 5000);
			TEST_ASSERT(gTransVacuum[1].Status.Blower.xMoving);
			nextState();
			break;

		case 14:
			strcpy(txStateDesc, "Testing alarm to stop");
			TEST_BUSY_CONDITION( gMachine.St.exec.fast < exTimesPreFast + 3 ); //We'll wait xx scan cycles
			gTransVacuum[1].Alarms.xAlrBlowersAnyCB = TRUE;
			nextState();
			break;

		case 15:
			TEST_BUSY_CONDITION(!gTransVacuum[1].Alarms.xAlrBlowersAnyCB);
			nextState();
			break;

		case 16:
			strcpy(txStateDesc, "BlowerStoppedW/Alarm");
			endtime=clock_ms();
			TEST_BUSY_CONDITION(endtime < TimeLast + 5000);
			TEST_ASSERT(!gTransVacuum[1].Status.Blower.xMoving);
			nextState();
			break;

		case 17: //stopping machine and returning to initial values
			strcpy(txStateDesc, "Returning to initial state");
			TEST_BUSY_CONDITION( gMachine.St.exec.fast < exTimesPreFast + 3 ); //We'll wait xx scan cycles
			gTransVacuum[1].Alarms.xAlrBlowersAnyCB = FALSE;
			gMachine.commandsSw.xStop_GI = TRUE;
			nextState();
			break;

		case 18:
			TEST_BUSY_CONDITION(!gMachine.St.Position.xInCap);
			gMachine.commandsSw.xReset_GI = TRUE;
			iTestState=0;

			TEST_DONE;
			break;

		default:
			break;

	}
}
_TEST test_StopBlowersWithAlarmByPass(void)
{
	strcpy(txTest, "test_StopBlowersWithAlarmByPass");
	switch (iTestState)
	{
		case 0:
			strcpy(txStateDesc, "Checking the blowers are installed");
			if (!gTransVacuum[1].Status.xInstalled){
			TEST_DONE;
			break;
			}

			else{
			strcpy(txStateDesc, "Going to ZERO");
			gSimMachine.Commands.xToZero = TRUE;
			nextState();
			break;
			}

		case 1:
			strcpy(txStateDesc, "Waiting the machine to be in Zero");
			TEST_BUSY_CONDITION( !gMachine.St.Mode.xZero );
			gTransVacuum[1].parSw.xActiveOutOfProduction = TRUE;
			gSimMachine.Commands.xToAuto = TRUE;
			nextState();
			break;

		case 2:
			strcpy(txStateDesc, "Waiting the machine to be in Auto and CAP");
			TEST_BUSY_CONDITION(!gMachine.St.Mode.xAuto);
			TEST_BUSY_CONDITION(!gMachine.St.Position.xInCap);
			gMachine.commandsSw.xReset_GI = TRUE;
			nextState();
			break;

		case 3:
			TEST_BUSY_CONDITION( gMachine.St.exec.fast < exTimesPreFast + 3 ); //We'll wait xx scan cycles
			gMachine.commandsSw.xToByPass_GI = TRUE;
			nextState();
			break;

		case 4:
			strcpy(txStateDesc, "TEST 2: ByPass");
			endtime = clock_ms();
			TEST_BUSY_CONDITION(endtime < TimeLast + 1000);
			nextState();
			break;

		case 5:
			strcpy(txStateDesc, "Giving xStart command");
			TEST_BUSY_CONDITION(!gMachine.St.AutoMode.xBypass); //We'll wait xx scan cycles
			gMachine.commandsSw.xStart_GI = TRUE;
			nextState();
			break;

		case 6: //checking if the machine reaches the positions it has to
			strcpy(txStateDesc, "Waiting for the start process to complete");
			TEST_BUSY_CONDITION(!gMachine.St.AutoMode.xProdORByPass);//averiguar cuales son las variables a comprobar
			TEST_BUSY_CONDITION(!gBelt.states.xRuningBelt);
			nextState();
			break;

		case 7:
			strcpy(txStateDesc, "BlowersStartInAOP");
			endtime=clock_ms();
			TEST_BUSY_CONDITION(endtime < TimeLast + 50);
			TEST_ASSERT(gTransVacuum[1].Status.Blower.rDutyCycle > 0);//de momento la condición no se cumple, revisar
			gTransVacuum[1].parSw.xActiveOutOfProduction = FALSE;
			nextState();
			break;

		case 8:
			TEST_BUSY_CONDITION(gTransVacuum[1].parSw.xActiveOutOfProduction);
			nextState();
			break;

		case 9:
			endtime=clock_ms();
			TEST_BUSY_CONDITION(endtime < TimeLast + 5000);
			//If the blowers are started by another functionality, do not consider the test Failed
			TEST_ASSERT(!gTransVacuum[1].Status.Blower.xMoving || gTransVacuum[1].Commands.xRunByLine || gTransVacuum[1].Commands.xRunByRemote);
			nextState();
			break;

		case 10:
			TEST_BUSY_CONDITION( gMachine.St.exec.fast < exTimesPreFast + 3 ); //We'll wait xx scan cycles
			gTransVacuum[1].parSw.xActiveOutOfProduction = TRUE;
			gMachine.commandsSw.xStart_GI = TRUE;
			nextState();
			break;

		case 11:
			TEST_BUSY_CONDITION(!gMachine.commandsSw.xStart_GI);
			TEST_BUSY_CONDITION(!gTransVacuum[1].parSw.xActiveOutOfProduction);
			nextState();
			break;

		case 12:
			endtime=clock_ms();
			TEST_BUSY_CONDITION(endtime < TimeLast + 5000);
			TEST_ASSERT(gTransVacuum[1].Status.Blower.xMoving);
			nextState();
			break;

		case 13:
			strcpy(txStateDesc, "Testing alarm to stop");
			TEST_BUSY_CONDITION( gMachine.St.exec.fast < exTimesPreFast + 3 ); //We'll wait xx scan cycles
			gTransVacuum[1].Alarms.xAlrBlowersAnyCB = TRUE;
			nextState();
			break;

		case 14:
			strcpy(txStateDesc, "BlowerStoppedW/Alarm");
			TEST_BUSY_CONDITION(!gTransVacuum[1].Alarms.xAlrBlowersAnyCB);
			nextState();
			break;

		case 15:
			endtime=clock_ms();
			TEST_BUSY_CONDITION(endtime < TimeLast + 5000);
			TEST_ASSERT(!gTransVacuum[1].Status.Blower.xMoving);
			nextState();
			break;

		case 16:
			strcpy(txStateDesc, "Returning to initial state");
			TEST_BUSY_CONDITION( gMachine.St.exec.fast < exTimesPreFast + 3 ); //We'll wait xx scan cycles
			gTransVacuum[1].Alarms.xAlrBlowersAnyCB = FALSE;
			gMachine.commandsSw.xStop_GI = TRUE;
			nextState();
			break;

		case 17:
			TEST_BUSY_CONDITION(!gMachine.St.Position.xInCap);
			gMachine.commandsSw.xReset_GI = TRUE;
			iTestState=0;

			TEST_DONE;
			break;

		default:
			break;

	}
}

/*
B+R UnitTest: This is generated code.
Do not edit! Do not move!
Description: UnitTest Testprogramm infrastructure (TestSet).
LastUpdated: 2023-04-26 09:55:10Z
By B+R UnitTest Helper Version: 2.0.1.59
*/
UNITTEST_FIXTURES(fixtures)
{
	new_TestFixture("test_StopBlowersOutProductionByPass", test_StopBlowersOutProductionByPass),
	new_TestFixture("test_StartBlowersOutProductionByPass", test_StartBlowersOutProductionByPass),
	new_TestFixture("test_StopBlowersOutProductionLab", test_StopBlowersOutProductionLab),
	new_TestFixture("test_StartBlowersOutProductionLab", test_StartBlowersOutProductionLab),
	new_TestFixture("test_StopBlowersWhenGoingOutOfManual", test_StopBlowersWhenGoingOutOfManual),
	new_TestFixture("test_StopBlowersWithAlarmLaboratory", test_StopBlowersWithAlarmLaboratory),
	new_TestFixture("test_StopBlowersWithAlarmByPass", test_StopBlowersWithAlarmByPass),
};

UNITTEST_CALLER_COMPLETE_EXPLICIT(TrVacuumTests, "TrVacuumTests", 0, 0, fixtures, 0, 0, 0);
```

#### TrVacuumTests.var - PVs for the program and test suite
```iecst
(********************************************************************
 * COPYRIGHT -- Bernecker + Rainer
 ********************************************************************
 * Program: TrVacuumTests
 * Author: Jorge Murria
 ********************************************************************
 * Local variables of program TrVacuumTests
 * General variables - do not change
 ********************************************************************)
(*Describe the test*)
VAR
	Testsuite : UtMgrTestSuite := (Name:='TrVacuumTests',Description:='Description of the Tests',Type:=utMgrTEST_TYPE_C,MetaInformation:='Some Meta Information can be added here');
END_VAR
(*Variables used in the tests*)
```

#### autoGeneratedFile.c - Auto generated code
```c
/*
B+R UnitTest: This is generated code.
Do not edit! Do not move!
Description: UnitTest Testprogramm infrastructure (List of TestSets).
LastUpdated: 2020-05-18 14:29:28Z
By B+R UnitTest Helper Version: 2.0.1.59
*/
#include "UnitTest.h"

UNITTEST_TESTSET_DECLARATION  TrVacuumTests;

UNITTEST_TESTSET_FIXTURES(utTestSets)
{
	new_TestSet(TrVacuumTests),
};
UNTITTEST_TESTSET_HANDLER();
```

### Program Logical/UnitTest/Tests/Cube (ANSIC)

#### autoGeneratedFile.c
```c
/*
B+R UnitTest: This is generated code.
Do not edit! Do not move!
Description: UnitTest Testprogramm infrastructure (List of TestSets).
LastUpdated: 2023-05-02 14:03:12Z
By B+R UnitTest Helper Version: 2.0.1.59
*/
#include "UnitTest.h"

UNITTEST_TESTSET_DECLARATION  Cube;

UNITTEST_TESTSET_FIXTURES(utTestSets)
{
	new_TestSet(Cube),
};
UNTITTEST_TESTSET_HANDLER();
```

#### Cube.c
```c
/********************************************************************
 * COPYRIGHT -- Bernecker + Rainer
 ********************************************************************
 * Program: ConsentsTests
 * Author: Jorge Murria
 ********************************************************************
 * Prepare machine with basic test to allow proper behabior
 * and starting tasks
 ********************************************************************/

#include <bur/plctypes.h>

#ifdef _DEFAULT_INCLUDES
#include <AsDefault.h>
#endif

#include "UnitTest.h"

#include <stdio.h>
#include <unistd.h>
#include <time.h>         /* clock_t, clock, CLOCKS_PER_SEC */

_LOCAL TIME TimeLast;
_LOCAL TIME endtime;
_LOCAL UDINT diff_t;
_LOCAL STRING stringAux[120];

#define FALSE 0
#define TRUE 1

void nextState(){
	exTimesPreFast = gMachine.St.exec.fast;
	exTimesPreSlow = gMachine.St.exec.slow;
	iTestState++;
	TimeLast = clock_ms();
	diff_t = diff_t;
	stringAux[120] = stringAux[120];
}

_TEST test_TestCase(void)
{
	strcpy(txTest, "test_TestCase");
	// Check txText <> than assigned, so just once
	if (strcmp(&txTest, &gSimMachine.Commands.LogTests.Text) != 0){
		strcpy(gSimMachine.Commands.LogTests.Text, txTest); gSimMachine.Commands.LogTests.xCommand = TRUE;
	}

	switch (iTestState)
	{
		case 0:
			gSimMachine.Commands.xToZero = TRUE;
			gSimThickCtrl.Commands.xEmptyMediaTracking = TRUE;
			nextState();
			break;

		case 1:
			strcpy(txStateDesc, "Waiting the machine to be in Zero");
			TEST_BUSY_CONDITION( gMachine.St.exec.fast < exTimesPreFast + 5 ); //We'll wait xx scan cycles

			endtime = clock_ms();
			TEST_BUSY_CONDITION( endtime < TimeLast + 500 ); //We'll wait xx ms

			TEST_BUSY_CONDITION( !gMachine.St.Mode.xZero );

			TEST_ASSERT(gMachine.St.Mode.xZero); //If variable is TRUE, the test is correct

			//This 2 lines just for the last TestCase
			strcpy(txTest, "test_TestCase Finished!! Congrats!");
			strcpy(txStateDesc, "--");

			iTestState = 0;
			TEST_DONE;

			nextState();
			break;

		default:
			break;
	}
}

_TEST test_StackReceiveUnexpectedMedia(void)
{
	if (!gThicknessCtrl.status.xNewMediaStackEnabled)
	{
		TEST_DONE;
	}

	TEST_BUSY_CONDITION( gMachine.St.exec.fast < exTimesPreFast + 10 ); //We'll wait xx scan cycles
	strcpy(txTest, "test_StackReceiveUnexpectedMedia");
	// Check txText <> than assigned, so just once
	if (strcmp(&txTest, &gSimMachine.Commands.LogTests.Text) != 0){
		strcpy(gSimMachine.Commands.LogTests.Text, txTest); gSimMachine.Commands.LogTests.xCommand = TRUE;
	}
	switch (iTestState)
	{
		case 0:
			gSimMachine.Commands.xToZero = TRUE;
			gMachine.commandsSw.xReset_GI = TRUE;
			gSimMachine.Parameters.Stack.xLoadNewMedia = FALSE;
			gSimThickCtrl.Commands.xEmptyMediaTracking = TRUE;
			nextState();
			break;

		case 1:
			strcpy(txStateDesc, "Going to Zero");
			TEST_BUSY_CONDITION( !gMachine.St.Mode.xZero );
			gSimMachine.Commands.xToAuto = TRUE;
			nextState();
			break;

		case 2:
			strcpy(txStateDesc, "Going to Auto");
			TEST_BUSY_CONDITION( !gMachine.St.Mode.xAuto );
			nextState();
			break;

		case 3:
			strcpy(txStateDesc, "Going to Production");
			TEST_BUSY_CONDITION( gMachine.St.exec.fast < exTimesPreFast + 3 ); //We'll wait xx scan cycles
			gSimMachine.Commands.xToProduction = TRUE;
			nextState();
			break;

		case 4:
			strcpy(txStateDesc, "Going to Print Position");
			TEST_BUSY_CONDITION( gMachine.St.exec.fast < exTimesPreFast + 3 ); //We'll wait xx scan cycles
			TEST_BUSY_CONDITION( !gMachine.St.Position.xInPrint );
			nextState();
			break;

		case 5:
			strcpy(txStateDesc, "Waiting the belt to start");
			TEST_BUSY_CONDITION( !gBelt.states.xRuningBelt);
			gSimMachine.Commands.Media.xContinuousMediaPresent = TRUE;
			TEST_BUSY_CONDITION( gMachine.St.exec.fast < exTimesPreFast + 5 ); //We'll wait xx scan cycles
			nextState();
			break;

		case 6:
			strcpy(txStateDesc, "Receiving media");
			TEST_BUSY_CONDITION( gMachine.St.exec.fast < exTimesPreFast + 3 ); //We'll wait xx scan cycles
			nextState();
			break;

		case 7:
			strcpy(txStateDesc, "Waiting the tray error to appear");
			endtime = clock_ms();
			if (gMachine.Al.Warning.xNotLoadedImage){
				nextState();
			}
			TEST_BUSY_CONDITION( endtime < TimeLast + 10000 ); //We'll wait xx ms
			nextState();
			break;

		case 8:
			TEST_ASSERT(gMachine.Al.Warning.xNotLoadedImage); //Alarm raised
			nextState();
			break;

		case 9:
			strcpy(txStateDesc, "Removing the error");
			gMachine.commandsSw.xReset_GI = TRUE;
			nextState();
			break;

		case 10:
			strcpy(txStateDesc, "Waiting the error to be removed");
			TEST_BUSY_CONDITION( gMachine.Al.Warning.xNotLoadedImage );
			gMachine.commandsSw.xReset_GI = FALSE;
			nextState();
			break;

		case 11:
			gSimMachine.Parameters.Stack.xLoadNewMedia = TRUE;

			iTestState = 0;

			strcpy(txTest, "test_StackReceiveUnexpectedMedia Finished!! Congrats!");
			strcpy(txStateDesc, "--");

			TEST_DONE;
			nextState();
			break;

		default:
			break;
	}
}

_TEST test_EnteringInAutoRemotely(void)
{
	// Do not execute the test if not machine controlled remotely
	if (!gMachine.Pt.xControlledRemotely)
	{
		TEST_DONE;
	}

	TEST_BUSY_CONDITION( gMachine.St.exec.fast < exTimesPreFast + 10 ); //We'll wait xx scan cycles
	strcpy(txTest, "test_EnteringInAutoRemotely");
	// Check txText <> than assigned, so just once
	if (strcmp(&txTest, &gSimMachine.Commands.LogTests.Text) != 0){
		strcpy(gSimMachine.Commands.LogTests.Text, txTest); gSimMachine.Commands.LogTests.xCommand = TRUE;
	}
	switch (iTestState)
	{
		case 0:
			gSimMachine.Commands.xToZero = TRUE;
			gSimThickCtrl.Commands.xEmptyMediaTracking = TRUE;
			nextState();
			break;

		case 1:
			strcpy(txStateDesc, "Going to Zero");
			TEST_BUSY_CONDITION( !gMachine.St.Mode.xZero );
			nextState();
			break;

		case 2:
			// Managing the selector
			gMachine.In.Buttons.xZero = FALSE;
			gMachine.In.Buttons.xManual = FALSE;
			gMachine.In.Buttons.xAuto = TRUE;

			// Raising the remot signal
			gMachine.commandsSw.xReset_GI = TRUE;

			strcpy(txStateDesc, "Going to Auto");

			nextState();
			break;

		case 3:

			TEST_BUSY_CONDITION( gMachine.St.exec.fast < exTimesPreFast + 10 ); //We'll wait xx scan cycles

			TEST_ASSERT(gMachine.St.Mode.xAuto); //If variable is TRUE, the test is correct

			iTestState = 0;

			strcpy(txTest, "test_EnteringInAutoRemotely Finished!! Congrats!");
			strcpy(txStateDesc, "--");

			TEST_DONE;
			nextState();
			break;

		default:
			break;
	}
}

_TEST test_Beeping1sec(void)
{
	// Do not execute the test if not machine controlled remotely
	if (!gMachine.Pt.xControlledRemotely)
	{
		TEST_DONE;
	}

	TEST_BUSY_CONDITION( gMachine.St.exec.fast < exTimesPreFast + 10 ); //We'll wait xx scan cycles
	strcpy(txTest, "test_Beeping1sec");
	// Check txText <> than assigned, so just once
	if (strcmp(&txTest, &gSimMachine.Commands.LogTests.Text) != 0){
		strcpy(gSimMachine.Commands.LogTests.Text, txTest); gSimMachine.Commands.LogTests.xCommand = TRUE;
	}
	switch (iTestState)
	{
		case 0:
			gSimMachine.Commands.xToZero = TRUE;
			gSimThickCtrl.Commands.xEmptyMediaTracking = TRUE;
			nextState();
			break;

		case 1:
			strcpy(txStateDesc, "Waiting to be in Zero");
			TEST_BUSY_CONDITION( !gMachine.St.Mode.xZero );
			gSimMachine.Commands.xToAuto = TRUE;
			nextState();
			break;

		case 2:
			strcpy(txStateDesc, "Going to Auto");
			TEST_BUSY_CONDITION( !gMachine.St.Mode.xAuto );
			nextState();
			break;

		case 3:
			strcpy(txStateDesc, "Going to Production");
			TEST_BUSY_CONDITION( gMachine.St.exec.fast < exTimesPreFast + 3 ); //We'll wait xx scan cycles
			gSimMachine.Commands.xToProduction = TRUE;
			nextState();
			break;

		case 4:
			strcpy(txStateDesc, "Going to Print Position");
			TEST_BUSY_CONDITION( gMachine.St.exec.fast < exTimesPreFast + 3 ); //We'll wait xx scan cycles
			nextState();
			break;

		case 5:
			strcpy(txStateDesc, "Waiting the belt to receive order to start");
			TEST_BUSY_CONDITION( !gBelt.commands.xRunBelt);
			nextState();
			break;

		case 6:
			strcpy(txStateDesc, "Waiting time to check Belt started");
			endtime = clock_ms();
			// Wait 1.5sec to review the status of the belt
			TEST_BUSY_CONDITION( endtime < TimeLast + 1500 ); //We'll wait xx ms
			TEST_ASSERT(gBelt.states.xRuningBelt); //Alarm raised
			nextState();
			break;

		case 7:
			iTestState = 0;

			strcpy(txTest, "test_Beeping1sec Finished!! Congrats!");
			strcpy(txStateDesc, "--");

			TEST_DONE;
			nextState();
			break;

		default:
			break;
	}
}

_TEST test_EnteringAndJogJamRecovery(void)
{
	// Do not execute the test if not jam recovery allowed
	if (!gMachine.Pt.xAllowJamRecovery)
	{
		TEST_DONE;
	}

	TEST_BUSY_CONDITION( gMachine.St.exec.fast < exTimesPreFast + 10 ); //We'll wait xx scan cycles
	strcpy(txTest, "test_EnteringAndJogJamRecovery");
	// Check txText <> than assigned, so just once
	if (strcmp(&txTest, &gSimMachine.Commands.LogTests.Text) != 0){
		strcpy(gSimMachine.Commands.LogTests.Text, txTest); gSimMachine.Commands.LogTests.xCommand = TRUE;
	}
	switch (iTestState)
	{
		case 0:
			gSimMachine.Commands.xToZero = TRUE;
			gSimThickCtrl.Commands.xEmptyMediaTracking = TRUE;
			nextState();
			break;

		case 1:
			strcpy(txStateDesc, "Waiting to be in Zero");
			TEST_BUSY_CONDITION( !gMachine.St.Mode.xZero );
			gSimMachine.Commands.xToAuto = TRUE;
			nextState();
			break;

		case 2:
			strcpy(txStateDesc, "Going to Auto");
			TEST_BUSY_CONDITION( gMachine.St.exec.slow < exTimesPreSlow + 3 ); //We'll wait xx scan cycles
			TEST_BUSY_CONDITION( !gMachine.St.Mode.xAuto );
			gMachine.commandsSw.xToJamRecovery = TRUE;
			nextState();
			break;

		case 3:
			strcpy(txStateDesc, "Going to Jam Recovery");
			TEST_BUSY_CONDITION( gMachine.St.exec.slow < exTimesPreSlow + 3 ); //We'll wait xx scan cycles
			TEST_BUSY_CONDITION( !gMachine.St.AutoMode.xJamRecovery );
			nextState();
			break;

		case 4:
			strcpy(txStateDesc, "Waiting to Be ready to jog");
			TEST_BUSY_CONDITION( gMachine.St.exec.slow < exTimesPreSlow + 3 ); //We'll wait xx scan cycles
			TEST_BUSY_CONDITION( !gMachine.St.Remote.xReadyToJogInJamRecovery );
			gMachine.In.xRemoteJog = TRUE;
			nextState();
			break;

		case 5:
			strcpy(txStateDesc, "Waiting the belt to start");
			TEST_BUSY_CONDITION( gMachine.St.exec.fast < exTimesPreFast + 3 ); //We'll wait xx scan cycles
			TEST_BUSY_CONDITION( !gBelt.states.xRuningBelt);
			TEST_ASSERT( gBelt.states.xRuningBelt); //(gBelt.states.rCurrentSpeed > 1 );
			gMachine.In.xRemoteJog = FALSE;
			nextState();
			break;

		case 6:
			strcpy(txStateDesc, "Waiting to stop the Belt");
			TEST_BUSY_CONDITION( gMachine.St.exec.fast < exTimesPreFast + 3 ); //We'll wait xx scan cycles
			TEST_ASSERT( !gBelt.states.xRuningBelt );
			nextState();
			break;

		case 7:
			gSimMachine.Commands.xToZero = TRUE;
			nextState();
			break;

		case 8:
			strcpy(txStateDesc, "Waiting to be in Zero");
			TEST_BUSY_CONDITION( !gMachine.St.Mode.xZero );

			iTestState = 0;

			strcpy(txTest, "test_EnteringAndJogJamRecovery Finished!! Congrats!");
			strcpy(txStateDesc, "--");

			TEST_DONE;
			nextState();
			break;

		default:
			break;
	}
}

_TEST test_NotJogIfNotJamRecovery(void)
{
	// Do not execute the test if not jam recovery allowed
	if (!gMachine.Pt.xAllowJamRecovery)
	{
		TEST_DONE;
	}

	TEST_BUSY_CONDITION( gMachine.St.exec.slow < exTimesPreSlow + 3 ); //We'll wait xx scan cycles
	strcpy(txTest, "test_NotJogIfNotJamRecovery");
	// Check txText <> than assigned, so just once
	if (strcmp(&txTest, &gSimMachine.Commands.LogTests.Text) != 0){
		strcpy(gSimMachine.Commands.LogTests.Text, txTest); gSimMachine.Commands.LogTests.xCommand = TRUE;
	}
	switch (iTestState)
	{
		case 0:
			gSimMachine.Commands.xToZero = TRUE;
			gSimThickCtrl.Commands.xEmptyMediaTracking = TRUE;
			nextState();
			break;

		case 1:
			strcpy(txStateDesc, "Waiting to be in Zero");
			TEST_BUSY_CONDITION( !gMachine.St.Mode.xZero );
			gSimMachine.Commands.xToAuto = TRUE;
			nextState();
			break;

		case 2:
			strcpy(txStateDesc, "Going to Auto");
			TEST_BUSY_CONDITION( gMachine.St.exec.slow < exTimesPreSlow + 3 ); //We'll wait xx scan cycles
			TEST_BUSY_CONDITION( !gMachine.St.Mode.xAuto );
			nextState();
			break;

		case 3:
			strcpy(txStateDesc, "Activating the jog");
			TEST_BUSY_CONDITION( gMachine.St.exec.slow < exTimesPreSlow + 3 ); //We'll wait xx scan cycles
			gMachine.In.xRemoteJog = TRUE;
			nextState();
			break;

		case 4:
			strcpy(txStateDesc, "Waiting the belt to start");
			TEST_BUSY_CONDITION( gMachine.St.exec.fast < exTimesPreFast + 3 ); //We'll wait xx scan cycles
			TEST_ASSERT( gBelt.states.rCurrentSpeed < 0.1 );
			gMachine.In.xRemoteJog = FALSE;
			nextState();
			break;

		case 5:
			gSimMachine.Commands.xToZero = TRUE;
			nextState();
			break;

		case 6:
			strcpy(txStateDesc, "Waiting to be in Zero");
			TEST_BUSY_CONDITION( !gMachine.St.Mode.xZero );

			iTestState = 0;

			strcpy(txTest, "test_NotJogIfNotJamRecovery Finished!! Congrats!");
			strcpy(txStateDesc, "--");

			TEST_DONE;
			nextState();
			break;

		default:
			break;
	}
}

/*
B+R UnitTest: This is generated code.
Do not edit! Do not move!
Description: UnitTest Testprogramm infrastructure (TestSet).
LastUpdated: 2023-05-22 09:37:32Z
By B+R UnitTest Helper Version: 2.0.1.59
*/
UNITTEST_FIXTURES(fixtures)
{
	new_TestFixture("test_TestCase", test_TestCase),
	new_TestFixture("test_StackReceiveUnexpectedMedia", test_StackReceiveUnexpectedMedia),
	new_TestFixture("test_EnteringInAutoRemotely", test_EnteringInAutoRemotely),
	new_TestFixture("test_Beeping1sec", test_Beeping1sec),
	new_TestFixture("test_EnteringAndJogJamRecovery", test_EnteringAndJogJamRecovery),
	new_TestFixture("test_NotJogIfNotJamRecovery", test_NotJogIfNotJamRecovery),
};

UNITTEST_CALLER_COMPLETE_EXPLICIT(Cube, "Cube", 0, 0, fixtures, 0, 0, 0);
```

- Program Logical/UnitTest/Tests/LineTests (ANSIC) (no source held here)

### Program Logical/UnitTest/Tests/FunctionsTests (ANSIC)
